# B&R Automation Studio project Lecture_09_jbl
Automation Studio 4.8.2.72

## Configuration Config1

### Task classes (Cpu.sw)
```
Cyclic#4:
  CarAlarm <- CarAlarm.prg
  Program <- Program.prg
```

## Logical view

### Program Logical/Program

#### Variables.var
```iecst
VAR
	castate : CARALARM;
	diSensorVibration : BOOL;
	diRemote : BOOL;
	doSiren : BOOL;
END_VAR
```

#### Main.st
```iecst
PROGRAM _INIT
	(* Insert code here *)

END_PROGRAM

PROGRAM _CYCLIC
	// Tilstandsskiftlogik / state change logic
	CASE castate OF
		CARALARM_DISARMED:
			IF diRemote THEN
				castate := CARALARM_ARMED;
			END_IF

		CARALARM_ARMED:
			IF diRemote THEN
				castate := CARALARM_DISARMED;
			ELSIF diSensorVibration THEN
				castate := CARALARM_INTRUSION;
			END_IF

		CARALARM_INTRUSION:
			IF diRemote THEN
				castate := CARALARM_DISARMED;
			END_IF

	END_CASE

	// Output logic
	CASE castate OF
		CARALARM_DISARMED:
			doSiren := FALSE;

		CARALARM_ARMED:

		CARALARM_INTRUSION:
			doSiren := TRUE;
	END_CASE

END_PROGRAM

PROGRAM _EXIT
	(* Insert code here *)

END_PROGRAM
```
